// TIA Portal V17 export
// export: Created 2023-02-14T02:49:30.976465Z, ExportSetting WithDefaults, DisplayName Totally Integrated Automation Portal, DisplayVersion V17, DisplayName TIA Portal Openness, DisplayVersion V17, DisplayName TIA Portal Teamcenter Gateway, DisplayVersion V17, DisplayName TIA Portal Version Control Interface, DisplayVersion V17, DisplayName SINAMICS Startdrive Advanced, DisplayVersion V17, DisplayName SINAMICS Startdrive G130, G150, S120, S150, SINAMICS MV, S210, DisplayVersion V17, DisplayName SINAMICS Startdrive G110M, G120, G120C, G120D, G120P, G115D, DisplayVersion V17, DisplayName STEP 7 Professional, DisplayVersion V17, DisplayName STEP 7 Safety, DisplayVersion V17, DisplayName WinCC Professional, DisplayVersion V17
DATA_BLOCK "IO Analog Storage_DB"   // DB9
VERSION : 0.1
// stored: AutoNumber true, DBAccessibleFromOPCUA true, DBAccessibleFromWebserver true, InstanceOfName IO Analog Storage, InstanceOfType FB
"IO Analog Storage"
   // VAR_INPUT
   //    Init : Bool;
   //    Reset : Bool;
   // END_VAR
   // VAR
   //    "LT-23.01" : "Ana_w_K1K2";
   //    "LT-24.01" : "Ana_w_K1K2";
   //    "LT-33.01" : "Ana_w_K1K2";
   //    "LT-34.01" { S7_SetPoint := 'True'} : "Ana_w_K1K2";
   //    "LT-35.01" { S7_SetPoint := 'True'} : "Ana_w_K1K2";
   //    "LT-79.01" { S7_SetPoint := 'True'} : "Ana_w_K1K2";
   //    "LT-81.01" { S7_SetPoint := 'True'} : "Ana_w_K1K2";
   //    "LT-84.01" { S7_SetPoint := 'True'} : "Ana_w_K1K2";
   //    "LT-82.01" { S7_SetPoint := 'True'} : "Ana_w_K1K2";
   // END_VAR
BEGIN
END_DATA_BLOCK
